Yaskawa INFORM job: X2_57-69(1)(90,0).JBI

/JOB
//NAME X2_57-69(1)(90,0)
//POS
///NPOS 359,359,359,20,0,0
///TOOL 0
///POSTYPE PULSE
///PULSE
C00000=1941,-102693,-129564,10,101994,-18
C00001=-114160,-110711,-132276,13468,99543,32658
C00002=-115352,64839,21503,33302,71092,28193
C00003=-108531,78392,43986,16123,55140,37786
C00004=-108866,85252,55178,17040,51979,37122
C00005=-108996,88365,60166,17472,50599,36819
C00006=-108995,88536,62039,17737,49581,36632
C00007=-109034,88718,61766,17697,49840,36662
C00008=-109565,92254,66229,18307,49070,36272
C00009=-109034,88718,61766,17697,49840,36662
C00010=-108904,85509,56654,17244,51243,36976
C00011=-108571,78466,45235,16289,54445,37659
C00012=-107997,64928,29160,15382,57165,38310
C00013=-122208,49017,56535,29995,44799,-20500
C00014=-121054,58896,69591,30976,41821,-21001
C00015=-120607,61403,73283,31313,40811,-21157
C00016=-120607,63170,76793,32085,39739,-21613
C00017=-120607,62274,75028,31694,40274,-21383
C00018=-120608,64965,78215,32056,39778,-21596
C00019=-120607,62274,75028,31694,40274,-21383
C00020=-121364,56707,67057,30894,42308,-20982
C00021=-122534,47142,54464,30007,45185,-20534
C00022=-121995,48000,54847,25969,42983,-17450
C00023=-121016,58047,68030,26856,40021,-17900
C00024=-120639,62684,74202,27406,38635,-18182
C00025=-120639,64991,78769,28376,37190,-18734
C00026=-120639,62684,74202,27406,38635,-18182
C00027=-120856,61874,74409,27857,38220,-18464
C00028=-120445,66454,79858,28202,37199,-18614
C00029=-120856,61874,74409,27857,38220,-18464
C00030=-121238,57224,68232,27288,39602,-18174
C00031=-122229,47153,55046,26369,42553,-17714
C00032=-125892,1211,1187,22441,56600,-15676
C00033=-137814,-110158,-69296,24031,60757,-19595
C00034=-137728,-112604,-73316,23755,61850,-19313
C00035=-105364,-57557,-72999,2137,103390,46474
C00036=-118914,16972,-18491,2200,108489,41969
C00037=-119887,15858,-15574,2165,106148,41596
C00038=-121510,15333,-13660,2144,104740,41021
C00039=-121541,15180,-12957,2137,104232,41000
C00040=-120276,15500,-14332,2152,105210,41447
C00041=-120275,15157,-12943,2141,104179,41429
C00042=-120845,15149,-12950,2139,104194,41236
C00043=-120275,15157,-12943,2141,104179,41429
C00044=-120276,15500,-14332,2152,105210,41447
C00045=-118914,16972,-18491,2200,108489,41969
C00046=-118859,16942,-18519,2200,108489,41988
C00047=-119832,15826,-15604,2165,106148,41615
C00048=-121413,15318,-13781,2144,104807,41053
C00049=-121413,15142,-12992,2137,104231,41043
C00050=-120221,15467,-14363,2153,105210,41465
C00051=-120221,15224,-12881,2141,104174,41447
C00052=-120790,15216,-12889,2139,104189,41254
C00053=-120221,15224,-12881,2141,104174,41447
C00054=-120221,15467,-14363,2153,105210,41465
C00055=-118859,16942,-18519,2200,108489,41988
C00056=-102402,-48698,-67991,2144,104784,47502
C00057=-177118,-86899,-49314,70294,69346,55717
C00058=-162665,-62437,-38431,68363,61957,60420
C00059=-158949,-60049,-34374,68890,58994,60353
C00060=-157479,-59004,-32692,69121,57826,60324
C00061=-157483,-57954,-30366,69642,57492,59876
C00062=-157504,-58291,-30998,69516,57587,59981
C00063=-155795,-59629,-31689,69630,56353,60099
C00064=-157504,-58291,-30998,69516,57587,59981
C00065=-157484,-58197,-30924,69514,57575,59985
C00066=-156523,-55844,-29677,69224,57103,60350
C00067=-157484,-58197,-30924,69514,57575,59985
C00068=-162670,-61686,-36716,68690,61698,60098
C00069=-161856,-67053,-41033,60813,38521,63477
C00070=-158996,-62210,-35558,60803,36300,63693
C00071=-157898,-60236,-33315,60834,35435,63760
C00072=-157901,-59173,-30986,61942,34994,63152
C00073=-156769,-58533,-30874,61190,34419,63655
C00074=-156166,-58108,-30651,60848,34087,63889
C00075=-156769,-58791,-31436,60917,34526,63803
C00076=-161883,-66170,-39058,61667,38156,62985
C00077=-175307,-91794,-54277,68294,45083,57713
C00078=-192656,-55134,-37587,64210,60039,59083
C00079=-162159,-23717,-10104,69718,77823,43469
C00080=-159534,-21701,-5637,70155,75421,43047
C00081=-158490,-20805,-3772,70360,74468,42873
C00082=-158493,-19842,-1317,70611,74104,42419
C00083=-158430,-19960,-1760,70561,74138,42521
C00084=-157077,-18912,-994,70615,73251,42719
C00085=-158430,-19960,-1760,70561,74138,42521
C00086=-162097,-22978,-8198,69866,77487,43129
C00087=-164656,-6441,2331,68796,80646,40119
C00088=-162354,-4355,7073,69146,78392,39620
C00089=-161441,-2725,10948,69469,77194,39063
C00090=-161443,-1987,12871,69626,76894,38710
C00091=-161439,-2551,11387,69503,77124,38984
C00092=-160415,-1923,12464,69637,76311,38965
C00093=-159548,-1589,12743,69678,75730,39076
C00094=-160719,-2768,10769,69490,76742,39193
C00095=-164702,-5497,5223,68969,80178,39553
C00096=-192656,-55134,-37587,64210,60039,59083
C00097=-125486,-104854,-75041,22917,86800,-65584
C00098=-126033,-92220,-87194,23391,99857,-63257
C00099=-126008,-87407,-69757,22927,92227,-64737
C00100=-122771,-89042,-67284,23124,89141,-64144
C00101=-121425,-89554,-66224,23215,87919,-63888
C00102=-121418,-87602,-63818,23218,87477,-63971
C00103=-121371,-87768,-64101,23220,87545,-63941
C00104=-119041,-87737,-64090,23370,86898,-63214
C00105=-121371,-87768,-64101,23220,87545,-63941
C00106=-119842,-88584,-64995,23320,87236,-63441
C00107=-119807,-91269,-65466,23334,86221,-63626
C00108=-119842,-88584,-64995,23320,87236,-63441
C00109=-121199,-88128,-66077,23230,88448,-63702
C00110=-124465,-86636,-68609,23034,91510,-64308
C00111=-142854,-85767,-72329,35934,81198,-48667
C00112=-140267,-86079,-63689,45810,58760,-32657
C00113=-135996,-80956,-60126,44498,56909,-31284
C00114=-134384,-78850,-58646,43955,56229,-30750
C00115=-134256,-77036,-56222,44175,55757,-30924
C00116=-134288,-77408,-56713,44133,55854,-30891
C00117=-132164,-77894,-56932,43544,54718,-30303
C00118=-134288,-77408,-56713,44133,55854,-30891
C00119=-88320,-91033,-56979,-46001,31828,15275
C00120=-89280,-88900,-56774,-44237,32046,14267
C00121=-88320,-91033,-56979,-46001,31828,15275
C00122=-85210,-101515,-62011,-50678,31900,18023
C00123=-89666,-105996,-71374,-46997,57370,39665
C00124=-112926,-92756,-65130,-39557,61499,44934
C00125=-117841,-88867,-61535,-38560,59130,43528
C00126=-119732,-87223,-60045,-38129,58240,42969
C00127=-119742,-85223,-57591,-38309,57852,43124
C00128=-119765,-85676,-58172,-38256,57941,43076
C00129=-121812,-86923,-58375,-37936,56635,42605
C00130=-119765,-85676,-58172,-38256,57941,43076
C00131=-121275,-85554,-58782,-37706,57631,42461
C00132=-122404,-83336,-58379,-37071,57860,41818
C00133=-121275,-85554,-58782,-37706,57631,42461
C00134=-114616,-91226,-63955,-39185,60786,44412
C00135=-114645,-97965,-79407,-37345,65578,42515
C00136=-116729,-83918,-76551,-18553,86191,61698
C00137=-117159,-89242,-76095,-11181,89587,70256
C00138=-119083,-90759,-73003,-11190,86687,69852
C00139=-119889,-89726,-70248,-11201,85432,69686
C00140=-119897,-88175,-68603,-11203,85218,69702
C00141=-119889,-89726,-70248,-11201,85432,69686
C00142=-119873,-91603,-70614,-11208,84708,69757
C00143=-119889,-89726,-70248,-11201,85432,69686
C00144=-107060,-93796,-69139,-19617,83326,67746
C00145=-109561,-94345,-69347,-19648,82582,66969
C00146=-107060,-93796,-69139,-19617,83326,67746
C00147=-120981,-91693,-72872,-11196,85873,69270
C00148=-118990,-90334,-76042,-11186,88750,69699
C00149=-119015,-93571,-89875,-11280,95471,69085
C00150=-121827,-98987,-110994,4235,90756,33976
C00151=-126467,-111869,-98615,30475,51467,-26148
C00152=-122938,-103029,-94111,27808,51796,-24337
C00153=-121643,-99583,-92275,26825,51945,-23680
C00154=-121634,-97826,-90039,26985,51518,-23798
C00155=-121643,-99583,-92275,26825,51945,-23680
C00156=-130783,-80407,-84869,35916,67887,-27578
C00157=-128717,-80853,-85070,35145,66956,-27002
C00158=-130783,-80407,-84869,35916,67887,-27578
C00159=-107674,-109601,-92730,7088,37825,-14001
C00160=-108083,-105924,-92018,7248,39302,-14088
C00161=-107674,-109601,-92730,7088,37825,-14001
C00162=-110011,-124661,-99237,10171,34381,-15732
C00163=-126906,-107253,-113226,22382,79753,-37979
C00164=-126893,-93432,-102362,29867,101882,-55415
C00165=-122864,-96655,-100816,29402,98217,-54829
C00166=-121215,-97700,-100096,29236,96792,-54563
C00167=-121210,-96197,-97952,29195,96310,-54685
C00168=-121215,-97700,-100096,29236,96792,-54563
C00169=-121163,-96448,-98340,29200,96390,-54646
C00170=-118846,-96389,-98319,29071,95614,-53959
C00171=-121163,-96448,-98340,29200,96390,-54646
C00172=-120263,-97948,-99498,29148,96030,-54394
C00173=-120240,-102374,-100607,29046,94623,-54741
C00174=-120263,-97948,-99498,29148,96030,-54394
C00175=-125973,-93962,-101877,29758,101067,-55277
C00176=-118596,-129181,-126473,-9366,77401,-2206
C00177=-114435,-108672,-97735,-33612,57488,30842
C00178=-118529,-101099,-93472,-31282,56999,29098
C00179=-120051,-98101,-91728,-30387,56847,28447
C00180=-120058,-96382,-89499,-30544,56421,28577
C00181=-120051,-98101,-91728,-30387,56847,28447
C00182=-120087,-96650,-89858,-30501,56482,28544
C00183=-122421,-96636,-89851,-29327,55655,27727
C00184=-120087,-96650,-89858,-30501,56482,28544
C00185=-120936,-97217,-90733,-29999,56393,28182
C00186=-120939,-93406,-89800,-29561,57600,27814
C00187=-120936,-97217,-90733,-29999,56393,28182
C00188=-115418,-107792,-96770,-33217,56982,30555
C00189=-105146,-130010,-122753,-24377,88875,54529
C00190=-114428,-145611,-119705,-15408,97435,71230
C00191=-117464,-150573,-117642,-15685,93169,70698
C00192=-118771,-152166,-116683,-15828,91559,70446
C00193=-118800,-148516,-114162,-15837,91865,70397
C00194=-118771,-152166,-116683,-15828,91559,70446
C00195=-89023,-160145,-112498,-25773,88935,79257
C00196=-92598,-162169,-112911,-26414,87133,78351
C00197=-89023,-160145,-112498,-25773,88935,79257
C00198=-143634,-123316,-108912,-7172,105756,63537
C00199=-144414,-127929,-109749,-7250,103844,63374
C00200=-143634,-123316,-108912,-7172,105756,63537
C00201=-142718,-121013,-109514,-7059,107379,63770
C00202=-140567,-114497,-110685,-6827,111603,64303
C00203=-106156,-132360,-130153,-17350,90664,54849
C00204=-113451,-107662,-104229,-36971,70393,33800
C00205=-118206,-101735,-100389,-35240,68968,32234
C00206=-120007,-99320,-98805,-34543,68461,31631
C00207=-120014,-97721,-96632,-34652,68030,31771
C00208=-120007,-99320,-98805,-34543,68461,31631
C00209=-120011,-97828,-96896,-34630,68120,31742
C00210=-122349,-97818,-96890,-33771,67193,31043
C00211=-120011,-97828,-96896,-34630,68120,31742
C00212=-121054,-97492,-97790,-34094,68307,31234
C00213=-121054,-93214,-96669,-33787,69569,30828
C00214=-121054,-97492,-97790,-34094,68307,31234
C00215=-114636,-105862,-103272,-36519,70163,33365
C00216=-114279,-101889,-100082,-25331,80876,44864
C00217=-118566,-99424,-96391,-24445,78685,43735
C00218=-120245,-97521,-93811,-24102,77637,43327
C00219=-120247,-96657,-92660,-24122,77395,43376
C00220=-120219,-96976,-93108,-24119,77505,43364
C00221=-122549,-96954,-93097,-23561,76842,42630
C00222=-120219,-96976,-93108,-24119,77505,43364
C00223=-114306,-100541,-98340,-25348,80523,44930
C00224=-120621,-97394,-101621,-24202,63073,45941
C00225=-120621,-97613,-99404,-24510,61722,46250
C00226=-126885,-95808,-100508,-15136,62705,44325
C00227=-124891,-100138,-106487,-19050,76932,40471
C00228=-124330,-97085,-92322,-20020,71587,41486
C00229=-120096,-97587,-96517,-20033,105608,38386
C00230=-120621,-97666,-97219,-19653,110159,37614
C00231=-120621,-97564,-100279,-19942,111985,37290
C00232=-114267,-119022,-117316,-18586,97333,41934
C00233=-120586,-140068,-100376,-59799,22791,77658
C00234=-120585,-131836,-89399,-65340,21573,80326
C00235=-120301,-131910,-88922,-66286,21610,80804
C00236=-120198,-131934,-88749,-66625,21626,80975
C00237=-119916,-129593,-85873,-68118,21579,81715
C00238=-118482,-138777,-95380,-52510,29730,72880
C00239=-120255,-147562,-109916,-33672,49046,60189
C00240=-120254,-140089,-100414,-34669,47370,60868
C00241=-115468,-148569,-111904,-12737,99323,53877
C00242=-120588,-148294,-110670,-9262,106248,51768
C00243=-120588,-160541,-124626,-9395,108516,51590
C00244=-136842,-121669,-124376,16041,91150,-8624
C00245=-120606,-113410,-86554,36159,18075,-56282
C00246=-120605,-110678,-81352,39700,16640,-57934
C00247=-120584,-111701,-82271,39578,16661,-57878
C00248=-120580,-111920,-82466,39553,16665,-57867
C00249=-120605,-109556,-79302,41216,16112,-58638
C00250=-124077,-125780,-98632,32708,39047,-51685
C00251=-120496,-124050,-111043,24637,69959,-42697
C00252=-120664,-121871,-104765,25113,67511,-43309
C00253=-121671,-124094,-110510,20986,97112,-39569
C00254=-120608,-124256,-111795,20648,99670,-38855
C00255=-120609,-125131,-115147,20777,101183,-38590
C00256=-120610,-125783,-123647,21277,105768,-37763
C00257=-120668,-128769,-125921,-5871,89606,-827
C00258=-107053,-95803,-77707,-38578,68772,44507
C00259=-120618,-86239,-59568,-37363,57829,42393
C00260=-120528,-85716,-59123,-36997,58097,42691
C00261=-120619,-91352,-71155,-22510,73817,56639
C00262=-119738,-88100,-63683,-22964,71349,57460
C00263=-119548,-88867,-66660,-18371,78749,62657
C00264=-120622,-86591,-69531,-13569,88626,68335
C00265=-120425,-89920,-79314,-13611,92853,67941
C00266=-120620,-95688,-83779,-13612,92610,67900
C00267=-120653,-118153,-99445,8937,69074,27704
C00268=-120618,-86290,-59555,39610,31833,-26802
C00269=-120617,-83679,-54099,41791,30283,-27941
C00270=-120617,-83181,-53105,42201,30015,-28153
C00271=-120617,-83020,-52785,42335,29929,-28222
C00272=-120619,-93115,-75724,25664,64689,-43944
C00273=-120826,-86244,-59129,27057,59793,-46292
C00274=-121400,-88637,-64040,23275,84750,-62478
C00275=-120618,-88758,-64988,22876,88456,-64391
C00276=-120618,-90407,-68808,22886,89847,-64125
C00277=-120645,-96149,-85177,23134,96436,-62865
C00278=-120704,-139648,-98792,22953,83536,-65363
C00279=-201677,-83839,-16745,82551,61455,23328
C00280=-193287,-71994,-23753,71338,80116,26125
C00281=-188716,-68676,-18939,72756,76807,26050
C00282=-186807,-37234,2063,68557,93943,25131
C00283=-186791,-37375,1977,68560,93924,25125
C00284=-188875,-55332,-8770,71294,85660,29887
C00285=-186990,-46090,-3659,67979,93495,33535
C00286=-187169,-52287,-8326,67185,92343,33510
C00287=-188906,-62105,-11935,69333,88967,33384
C00288=-188683,-64142,-13243,69128,88603,33879
C00289=-187867,-62779,-12578,68415,90081,34352
C00290=-188794,-66315,-17993,66765,90030,34259
C00291=-197371,-61565,-20436,64467,96999,34726
C00292=-180892,-45026,-152,77390,64230,28169
C00293=-201677,-83839,-16745,82551,61455,23328
C00294=-102465,-98091,-57376,11154,53691,1192
C00295=-117523,-2788,-9530,25488,75365,-1139
C00296=-125139,57134,55592,35785,69072,-6421
C00297=-125133,64451,72830,37508,63513,-8429
C00298=-123932,76756,90632,38887,59314,-9544
C00299=-123464,84249,101464,39928,56909,-10353
C00300=-122296,71715,85090,35181,54513,-6915
C00301=-122189,68599,81314,33173,52324,-4280
C00302=-122589,68250,80867,31901,50792,-2732
C00303=-122908,67120,79438,30365,49475,-1044
C00304=-123218,66439,78655,28729,48083,651
C00305=-123718,66653,78885,28024,47440,1365
C00306=-121882,59213,71115,24134,43656,7775
C00307=-110842,52453,67135,-14467,33841,33723
C00308=-111073,52381,67059,-14368,33810,33647
C00309=-110346,48653,61790,-14496,35224,33792
C00310=-108666,36587,42456,-14007,41045,33643
C00311=-114621,109196,43725,31616,85766,30078
C00312=-108492,104701,44017,11484,73458,41705
C00313=-108890,108743,52585,11893,70378,41274
C00314=-108566,112524,59213,11878,68242,41168
C00315=-105655,126679,78153,10634,63557,41739
C00316=-105456,124563,73948,10396,65010,41943
C00317=-114621,109196,43725,31616,85766,30078
C00318=-117523,-2788,-9530,25488,75365,-1139
C00319=-102465,-98091,-57376,11154,53691,1192
C00320=-194924,-89332,-18186,86283,57168,22588
C00321=-189291,-99620,-43569,70052,49879,58298
C00322=-183385,-95654,-38841,71457,45923,58650
C00323=-179289,-94967,-37057,72626,43143,58783
C00324=-180541,-94166,-36956,72139,44032,58817
C00325=-181760,-88303,-31492,78702,40431,52425
C00326=-191947,-67176,-20621,75434,55592,47212
C00327=-188895,-71260,-14971,91913,47690,32624
C00328=-190378,-73018,-17241,90953,48654,32921
C00329=-194954,-78245,-22550,88961,51649,33203
C00330=-209629,-115340,-51402,66324,56026,36469
C00331=-117179,-93991,-70029,-10923,64438,-31948
C00332=-91116,-86743,-69135,-16598,71993,-23160
C00333=-103770,-45855,-47036,-2494,89723,45807
C00334=-105440,-45139,-42797,-2405,87433,45286
C00335=-105872,-44623,-40732,-2383,86415,45158
C00336=-107998,-22692,-26100,-2267,88615,44398
C00337=-107613,-23106,-28265,-2289,89747,44508
C00338=-106174,-23599,-32412,-2371,92085,44950
C00339=-103769,-45855,-47037,-2494,89723,45807
C00340=-105440,-45140,-42797,-2405,87433,45286
C00341=-105983,-45111,-40907,-2377,86269,45123
C00342=-108050,-23400,-26513,-2264,88505,44381
C00343=-107613,-23106,-28265,-2289,89747,44508
C00344=-106174,-23599,-32412,-2371,92085,44950
C00345=-106187,-23536,-40664,-2395,97191,44849
C00346=-112777,14050,-22213,-10109,94464,-2996
C00347=-124710,91382,43994,-20502,78853,-68751
C00348=-124710,90699,45107,-20567,77880,-68584
C00349=-124711,89465,47608,-20728,75840,-68228
C00350=-124762,93463,53735,-20858,74219,-67960
C00351=-124700,97572,58988,-20989,73184,-67752
C00352=-127201,90948,48694,-14686,76522,-68030
C00353=-125335,102453,72014,-19381,53758,-65341
C00354=-124858,91287,58679,-21278,49111,-64908
C00355=-124711,88619,50210,-21147,50008,-65361
C00356=-120351,15313,-32439,-6340,69848,-64116
C00357=-119749,-104989,-49747,-18878,19546,-56964
C00358=1074,-84890,-111921,820,92639,-133
BC00000=210618,668760,578653
BC00001=307087,668760,191900
BC00002=307087,789553,191900
BC00003=307087,789553,191900
BC00004=307087,789553,191900
BC00005=307087,789553,191900
BC00006=307087,789553,191900
BC00007=307087,789553,191900
BC00008=307087,789553,191900
BC00009=307087,789553,191900
BC00010=307087,789553,191900
BC00011=307087,789553,191900
BC00012=307087,789553,191900
BC00013=319173,776954,280603
BC00014=319173,776954,280603
BC00015=319173,776954,280603
BC00016=319173,776954,280603
BC00017=319173,776954,280603
BC00018=319173,776954,280603
BC00019=319173,776954,280603
BC00020=319173,776954,280603
BC00021=319173,776954,280603
BC00022=324465,771616,271785
BC00023=324465,771616,271785
BC00024=324465,771616,271785
BC00025=324465,771616,271785
BC00026=324465,771616,271785
BC00027=324465,771616,271785
BC00028=324465,771616,271785
BC00029=324465,771616,271785
BC00030=324465,771616,271785
BC00031=324465,771616,271785
BC00032=324465,747237,368530
BC00033=324465,670069,674761
BC00034=169071,670069,459913
BC00035=137209,684775,182974
BC00036=137209,684775,182974
BC00037=137209,684775,182974
BC00038=137209,684775,182974
BC00039=137209,684775,182974
BC00040=137209,684775,182974
BC00041=137209,684775,182974
BC00042=137209,684775,182974
BC00043=137209,684775,182974
BC00044=137209,684775,182974
BC00045=137209,684775,182974
BC00046=136881,731969,182759
BC00047=136881,731969,182759
BC00048=136881,731969,182759
BC00049=136881,731969,182759
BC00050=136881,731969,182759
BC00051=136881,731969,182759
BC00052=136881,731969,182759
BC00053=136881,731969,182759
BC00054=136881,731969,182759
BC00055=136881,731969,182759
BC00056=136881,673536,182759
BC00057=33003,666220,204314
BC00058=33003,666220,204314
BC00059=33003,666220,204314
BC00060=33003,666220,204314
BC00061=33003,666220,204314
BC00062=33003,666220,204314
BC00063=33003,666220,204314
BC00064=33003,666220,204314
BC00065=33003,666220,204314
BC00066=33003,666220,204314
BC00067=33003,666220,204314
BC00068=33003,666220,204314
BC00069=48470,666220,217137
BC00070=48470,666220,217137
BC00071=48470,666220,217137
BC00072=48470,666220,217137
BC00073=48470,666220,217137
BC00074=48470,666220,217137
BC00075=48470,666220,217137
BC00076=48470,666220,217137
BC00077=48470,666220,217137
BC00078=48470,666220,217137
BC00079=15,666220,230034
BC00080=15,666220,230034
BC00081=15,666220,230034
BC00082=15,666220,230034
BC00083=15,666220,230034
BC00084=15,666220,230034
BC00085=15,666220,230034
BC00086=15,666220,230034
BC00087=15,666220,235835
BC00088=15,666220,235835
BC00089=15,666220,235835
BC00090=15,666220,235835
BC00091=15,666220,235835
BC00092=15,666221,235834
BC00093=15,666220,235835
BC00094=15,666220,235835
BC00095=15,666220,235835
BC00096=48470,666220,217137
BC00097=32831,670161,1075175
BC00098=32831,729596,1075175
BC00099=32831,729596,1075175
BC00100=32831,729596,1075175
BC00101=32831,729596,1075175
BC00102=32831,729596,1075175
BC00103=32831,729596,1075175
BC00104=32831,729596,1075175
BC00105=32831,729596,1075175
BC00106=32831,729596,1075175
BC00107=32831,729596,1075175
BC00108=32831,729596,1075175
BC00109=32831,729596,1075175
BC00110=32831,729596,1075175
BC00111=37728,721693,1075175
BC00112=41810,715107,1075175
BC00113=41810,715107,1075175
BC00114=41810,715107,1075175
BC00115=41810,715107,1075175
BC00116=41810,715107,1075175
BC00117=41810,715107,1075175
BC00118=41810,715107,1075175
BC00119=41810,715107,1075175
BC00120=41810,715107,1075175
BC00121=41810,715107,1075175
BC00122=41810,715107,1075175
BC00123=53876,706752,1075175
BC00124=60427,702216,1075175
BC00125=60427,702216,1075175
BC00126=60427,702216,1075175
BC00127=60427,702216,1075175
BC00128=60427,702216,1075175
BC00129=60427,702216,1075175
BC00130=60427,702216,1075175
BC00131=60427,702216,1075175
BC00132=60427,702216,1075175
BC00133=60427,702216,1075175
BC00134=60427,702216,1075175
BC00135=60427,702216,1075175
BC00136=46834,716034,1075175
BC00137=41397,721561,1075175
BC00138=41397,721561,1075175
BC00139=41397,721561,1075175
BC00140=41397,721561,1075175
BC00141=41397,721561,1075175
BC00142=41397,721561,1075175
BC00143=41397,721561,1075175
BC00144=41397,721561,1075175
BC00145=41397,721561,1075175
BC00146=41397,721561,1075175
BC00147=41397,721561,1075175
BC00148=41397,721561,1075175
BC00149=41397,721561,1075175
BC00150=77086,766277,1075175
BC00151=137161,841550,1075175
BC00152=137161,841550,1075175
BC00153=137161,841550,1075175
BC00154=137161,841550,1075175
BC00155=137161,841550,1075175
BC00156=137161,841550,1075175
BC00157=137161,841550,1075175
BC00158=137161,841550,1075175
BC00159=137161,841550,1075175
BC00160=137161,841550,1075175
BC00161=137161,841550,1075175
BC00162=137161,841550,1075175
BC00163=128673,864447,1075175
BC00164=121183,884651,1075175
BC00165=121183,884651,1075175
BC00166=121183,884651,1075175
BC00167=121183,884651,1075175
BC00168=121183,884651,1075175
BC00169=121183,884651,1075175
BC00170=121183,884651,1075175
BC00171=121183,884651,1075175
BC00172=121183,884651,1075175
BC00173=121183,884651,1075175
BC00174=121183,884651,1075175
BC00175=121183,884651,1075175
BC00176=162519,857645,1075175
BC00177=188050,840965,1075175
BC00178=188050,840965,1075175
BC00179=188050,840965,1075175
BC00180=188050,840965,1075175
BC00181=188050,840965,1075175
BC00182=188050,840965,1075175
BC00183=188050,840965,1075175
BC00184=188050,840965,1075175
BC00185=188050,840965,1075175
BC00186=188050,840965,1075175
BC00187=188050,840965,1075175
BC00188=188050,840965,1075175
BC00189=177981,881480,1075175
BC00190=169709,914761,1075175
BC00191=169709,914761,1075175
BC00192=169709,914761,1075175
BC00193=169709,914761,1075175
BC00194=169709,914761,1075175
BC00195=169709,914761,1075175
BC00196=169709,914761,1075175
BC00197=169709,914761,1075175
BC00198=169709,914761,1075175
BC00199=169709,914761,1075175
BC00200=169709,914761,1075175
BC00201=169709,914761,1075175
BC00202=169709,914761,1075175
BC00203=159152,880596,1075175
BC00204=150354,852125,1075175
BC00205=150354,852125,1075175
BC00206=150354,852125,1075175
BC00207=150354,852125,1075175
BC00208=150354,852125,1075175
BC00209=150354,852125,1075175
BC00210=150354,852125,1075175
BC00211=150354,852125,1075175
BC00212=150354,852125,1075175
BC00213=150354,852125,1075175
BC00214=150354,852125,1075175
BC00215=150354,852125,1075175
BC00216=138535,800539,1075175
BC00217=138535,800539,1075175
BC00218=138535,800539,1075175
BC00219=138535,800539,1075175
BC00220=138535,800539,1075175
BC00221=138535,800539,1075175
BC00222=138535,800539,1075175
BC00223=138535,800539,1075175
BC00224=139926,838224,1075175
BC00225=134477,841860,1075175
BC00226=132297,843314,1075175
BC00227=135301,861824,1075175
BC00228=135628,791701,1075175
BC00229=127557,845014,1075175
BC00230=128457,853081,1075175
BC00231=133547,854476,1075175
BC00232=133547,854476,1075175
BC00233=185526,847143,1075175
BC00234=185547,847145,1075175
BC00235=180367,852195,1075175
BC00236=178499,854016,1075175
BC00237=178499,854016,1075175
BC00238=181436,863252,1075175
BC00239=187425,882089,1075175
BC00240=187544,843803,1075173
BC00241=163075,924936,1075175
BC00242=160150,941259,1075175
BC00243=163894,945401,1075175
BC00244=155016,866117,1075175
BC00245=147551,828920,1075175
BC00246=147562,828921,1075175
BC00247=152516,835936,1075175
BC00248=153570,837428,1075175
BC00249=153570,837428,1075175
BC00250=143866,860842,1075175
BC00251=131316,891124,1075175
BC00252=131456,861099,1075175
BC00253=136555,907393,1075175
BC00254=134846,911418,1075175
BC00255=129544,912127,1075175
BC00256=129523,912125,1075175
BC00257=99118,813312,1075175
BC00258=64307,700180,1075175
BC00259=58098,703250,1075175
BC00260=55325,704971,1075175
BC00261=41598,728447,1075175
BC00262=60495,698876,1075175
BC00263=53827,709917,1075175
BC00264=47010,724325,1075175
BC00265=50143,727052,1075175
BC00266=50122,727050,1075175
BC00267=43900,716168,1075175
BC00268=35524,701519,1075175
BC00269=35534,701520,1075175
BC00270=39202,708199,1075175
BC00271=40669,710870,1075175
BC00272=31604,749687,1075172
BC00273=32090,681060,1075175
BC00274=35435,723771,1075175
BC00275=34090,730815,1075175
BC00276=29574,733664,1075175
BC00277=29574,733664,1075175
BC00278=29574,668853,1075175
BC00279=15,675786,401985
BC00280=15,747285,294679
BC00281=15,747285,294679
BC00282=15,747285,294679
BC00283=15,747285,294679
BC00284=15,747285,294679
BC00285=15,747285,294679
BC00286=15,747285,294679
BC00287=15,747285,294679
BC00288=15,747285,294679
BC00289=15,747285,294679
BC00290=15,747285,294679
BC00291=15,747285,294679
BC00292=15,675786,401985
BC00293=15,675786,401985
BC00294=281438,669247,530529
BC00295=311998,746592,376004
BC00296=327524,785889,297495
BC00297=327524,785889,297495
BC00298=327524,785889,297495
BC00299=327524,785889,297495
BC00300=327524,785889,297495
BC00301=327524,785889,297495
BC00302=327524,785889,297495
BC00303=327524,785889,297495
BC00304=327524,785889,297495
BC00305=327524,785889,297495
BC00306=327524,785889,297495
BC00307=327524,785889,297495
BC00308=327524,785889,297495
BC00309=327524,785889,297495
BC00310=327524,785889,297495
BC00311=301537,784116,209
BC00312=301537,784116,209
BC00313=301537,784116,209
BC00314=301537,784116,209
BC00315=301537,784116,209
BC00316=301537,784116,209
BC00317=301537,784116,209
BC00318=311998,746592,376004
BC00319=281438,669247,530529
BC00320=28742,675786,401985
BC00321=69504,715923,290542
BC00322=69504,715923,290542
BC00323=69504,715923,290542
BC00324=69504,715923,290542
BC00325=69504,715923,290542
BC00326=69504,715923,290542
BC00327=69504,715923,290542
BC00328=69504,715923,290542
BC00329=69504,715923,290542
BC00330=69504,715923,290542
BC00331=108267,707570,269586
BC00332=108267,707570,269586
BC00333=115634,729988,290459
BC00334=115634,729988,290459
BC00335=115634,729988,290459
BC00336=115634,729988,290459
BC00337=115634,729988,290459
BC00338=115634,729988,290459
BC00339=115460,777038,290246
BC00340=115460,777038,290246
BC00341=115460,777038,290246
BC00342=115460,777038,290246
BC00343=115460,777038,290246
BC00344=115460,777038,290246
BC00345=115460,777038,290246
BC00346=136842,705148,185844
BC00347=166172,670726,41167
BC00348=166193,670728,53
BC00349=164826,672048,53
BC00350=164280,672575,53
BC00351=164280,672575,53
BC00352=163972,755654,53
BC00353=160957,747196,53
BC00354=159846,741879,53
BC00355=160544,735428,53
BC00356=166172,670726,41167
BC00357=166172,670726,387185
BC00358=166172,670726,387185
EC00000=798156,0
EC00001=798156,0
EC00002=798156,0
EC00003=798156,0
EC00004=798156,0
EC00005=798156,0
EC00006=798156,0
EC00007=798156,0
EC00008=798156,0
EC00009=798156,0
EC00010=798156,0
EC00011=798156,0
EC00012=798156,0
EC00013=798156,0
EC00014=798156,0
EC00015=798156,0
EC00016=798156,0
EC00017=798156,0
EC00018=798156,0
EC00019=798156,0
EC00020=798156,0
EC00021=798156,0
EC00022=798156,0
EC00023=798156,0
EC00024=798156,0
EC00025=798156,0
EC00026=798156,0
EC00027=798156,0
EC00028=798156,0
EC00029=798156,0
EC00030=798156,0
EC00031=798156,0
EC00032=798156,0
EC00033=798156,0
EC00034=798156,0
EC00035=798156,0
EC00036=798156,0
EC00037=798156,0
EC00038=798156,0
EC00039=798156,0
EC00040=798156,0
EC00041=798156,0
EC00042=798156,0
EC00043=798156,0
EC00044=798156,0
EC00045=798156,0
EC00046=798156,0
EC00047=798156,0
EC00048=798156,0
EC00049=798156,0
EC00050=798156,0
EC00051=798156,0
EC00052=798156,0
EC00053=798156,0
EC00054=798156,0
EC00055=798156,0
EC00056=798156,0
EC00057=798156,0
EC00058=798156,0
EC00059=798156,0
EC00060=798156,0
EC00061=798156,0
EC00062=798156,0
EC00063=798156,0
EC00064=798156,0
EC00065=798156,0
EC00066=798156,0
EC00067=798156,0
EC00068=798156,0
EC00069=798156,0
EC00070=798156,0
EC00071=798156,0
EC00072=798156,0
EC00073=798156,0
EC00074=798156,0
EC00075=798156,0
EC00076=798156,0
EC00077=798156,0
EC00078=798156,0
EC00079=798156,0
EC00080=798156,0
EC00081=798156,0
EC00082=798156,0
EC00083=798156,0
EC00084=798156,0
EC00085=798156,0
EC00086=798156,0
EC00087=798156,0
EC00088=798156,0
EC00089=798156,0
EC00090=798156,0
EC00091=798156,0
EC00092=798155,0
EC00093=798156,0
EC00094=798156,0
EC00095=798156,0
EC00096=798156,0
EC00097=975524,0
EC00098=975524,0
EC00099=975524,0
EC00100=975524,0
EC00101=975524,0
EC00102=975524,0
EC00103=975524,0
EC00104=975524,0
EC00105=975524,0
EC00106=975524,0
EC00107=975524,0
EC00108=975524,0
EC00109=975524,0
EC00110=975524,0
EC00111=975524,0
EC00112=975524,0
EC00113=975524,0
EC00114=975524,0
EC00115=975524,0
EC00116=975524,0
EC00117=975524,0
EC00118=975524,0
EC00119=975524,0
EC00120=975524,0
EC00121=975524,0
EC00122=975524,0
EC00123=975524,0
EC00124=975524,0
EC00125=975524,0
EC00126=975524,0
EC00127=975524,0
EC00128=975524,0
EC00129=975524,0
EC00130=975524,0
EC00131=975524,0
EC00132=975524,0
EC00133=975524,0
EC00134=975524,0
EC00135=975524,0
EC00136=975524,0
EC00137=975524,0
EC00138=975524,0
EC00139=975524,0
EC00140=975524,0
EC00141=975524,0
EC00142=975524,0
EC00143=975524,0
EC00144=975524,0
EC00145=975524,0
EC00146=975524,0
EC00147=975524,0
EC00148=975524,0
EC00149=975524,0
EC00150=975524,0
EC00151=975524,0
EC00152=975524,0
EC00153=975524,0
EC00154=975524,0
EC00155=975524,0
EC00156=975524,0
EC00157=975524,0
EC00158=975524,0
EC00159=975524,0
EC00160=975524,0
EC00161=975524,0
EC00162=975524,0
EC00163=975524,0
EC00164=975524,0
EC00165=975524,0
EC00166=975524,0
EC00167=975524,0
EC00168=975524,0
EC00169=975524,0
EC00170=975524,0
EC00171=975524,0
EC00172=975524,0
EC00173=975524,0
EC00174=975524,0
EC00175=975524,0
EC00176=975524,0
EC00177=975524,0
EC00178=975524,0
EC00179=975524,0
EC00180=975524,0
EC00181=975524,0
EC00182=975524,0
EC00183=975524,0
EC00184=975524,0
EC00185=975524,0
EC00186=975524,0
EC00187=975524,0
EC00188=975524,0
EC00189=975524,0
EC00190=975524,0
EC00191=975524,0
EC00192=975524,0
EC00193=975524,0
EC00194=975524,0
EC00195=975524,0
EC00196=975524,0
EC00197=975524,0
EC00198=975524,0
EC00199=975524,0
EC00200=975524,0
EC00201=975524,0
EC00202=975524,0
EC00203=975524,0
EC00204=975524,0
EC00205=975524,0
EC00206=975524,0
EC00207=975524,0
EC00208=975524,0
EC00209=975524,0
EC00210=975524,0
EC00211=975524,0
EC00212=975524,0
EC00213=975524,0
EC00214=975524,0
EC00215=975524,0
EC00216=975524,0
EC00217=975524,0
EC00218=975524,0
EC00219=975524,0
EC00220=975524,0
EC00221=975524,0
EC00222=975524,0
EC00223=975524,0
EC00224=975524,0
EC00225=975524,0
EC00226=975524,0
EC00227=975524,0
EC00228=975524,0
EC00229=975524,0
EC00230=975524,0
EC00231=975524,0
EC00232=975524,0
EC00233=975524,0
EC00234=975524,0
EC00235=975524,0
EC00236=975524,0
EC00237=975524,0
EC00238=975524,0
EC00239=975524,0
EC00240=975522,1
EC00241=975524,0
EC00242=975524,0
EC00243=975524,0
EC00244=975524,0
EC00245=975524,0
EC00246=975524,0
EC00247=975524,0
EC00248=975524,0
EC00249=975524,0
EC00250=975524,0
EC00251=975524,0
EC00252=975524,0
EC00253=975524,0
EC00254=975524,0
EC00255=975524,0
EC00256=975524,0
EC00257=975524,0
EC00258=975524,0
EC00259=975524,0
EC00260=975524,0
EC00261=975524,0
EC00262=975524,0
EC00263=975524,0
EC00264=975524,0
EC00265=975524,0
EC00266=975524,0
EC00267=975524,0
EC00268=975524,0
EC00269=975524,0
EC00270=975524,0
EC00271=975524,0
EC00272=975522,1
EC00273=975524,0
EC00274=975524,0
EC00275=975524,0
EC00276=975524,0
EC00277=975524,0
EC00278=975524,0
EC00279=798156,0
EC00280=798156,0
EC00281=798156,0
EC00282=798156,0
EC00283=798156,0
EC00284=798156,0
EC00285=798156,0
EC00286=798156,0
EC00287=798156,0
EC00288=798156,0
EC00289=798156,0
EC00290=798156,0
EC00291=798156,0
EC00292=798156,0
EC00293=798156,0
EC00294=798156,0
EC00295=798156,0
EC00296=798156,0
EC00297=798156,0
EC00298=798156,0
EC00299=798156,0
EC00300=798156,0
EC00301=798156,0
EC00302=798156,0
EC00303=798156,0
EC00304=798156,0
EC00305=798156,0
EC00306=798156,0
EC00307=798156,0
EC00308=798156,0
EC00309=798156,0
EC00310=798156,0
EC00311=798156,0
EC00312=798156,0
EC00313=798156,0
EC00314=798156,0
EC00315=798156,0
EC00316=798156,0
EC00317=798156,0
EC00318=798156,0
EC00319=798156,0
EC00320=798156,0
EC00321=798156,0
EC00322=798156,0
EC00323=798156,0
EC00324=798156,0
EC00325=798156,0
EC00326=798156,0
EC00327=798156,0
EC00328=798156,0
EC00329=798156,0
EC00330=798156,0
EC00331=798156,0
EC00332=798156,0
EC00333=798156,0
EC00334=798156,0
EC00335=798156,0
EC00336=798156,0
EC00337=798156,0
EC00338=798156,0
EC00339=798156,0
EC00340=798156,0
EC00341=798156,0
EC00342=798156,0
EC00343=798156,0
EC00344=798156,0
EC00345=798156,0
EC00346=798156,0
EC00347=798156,0
EC00348=798156,0
EC00349=798156,0
EC00350=798156,0
EC00351=798156,0
EC00352=798156,0
EC00353=798156,0
EC00354=798156,0
EC00355=798156,0
EC00356=798156,0
EC00357=798156,0
EC00358=798156,0
///POSTYPE BASE
///RECTAN
///RCONF 0,0,0,0,0,0,0,0,0,0,0,0,0,0,0,0,0,0,0,0,0,0,0,0
P00006=0.222,-3.123,-1.508,0.0000,0.0000,0.0000
P00020=2.715,4.999,8.452,0.0000,0.0000,0.0000
P00021=-0.225,-6.128,-0.405,0.0000,0.0000,0.0000
P00022=0.222,-3.123,-1.508,0.0000,0.0000,0.0000
P00023=0.143,-0.036,0.682,0.0000,0.0000,0.0000
P00024=0.145,-0.552,1.326,0.0000,0.0000,0.0000
P00025=-2.003,0.006,0.728,0.0000,0.0000,0.0000
P00026=0.562,-0.002,-0.337,0.0000,0.0000,0.0000
P00031=1.853,-0.001,-1.549,0.0000,0.0000,0.0000
P00032=1.957,0.503,-7.217,0.0000,0.0000,0.0000
///RCONF 0,0,0,0,1,0,0,0,0,0,0,0,0,0,0,0,0,0,0,0,0,0,0,0
P00033=-0.123,0.612,-5.012,0.0000,0.0000,0.0000
///RCONF 0,0,0,0,0,0,0,0,0,0,0,0,0,0,0,0,0,0,0,0,0,0,0,0
P00034=-0.304,0.773,-2.693,0.0000,0.0000,0.0000
P00035=2.817,0.591,-1.622,0.0000,0.0000,0.0000
P00036=-1.108,-0.829,1.850,0.0000,0.0000,0.0000
P00037=0.023,0.937,-2.677,0.0000,0.0000,0.0000
P00038=0.158,-1.133,-1.952,0.0000,0.0000,0.0000
P00039=0.012,-3.081,-0.106,0.0000,0.0000,0.0000
P00040=-0.030,9.648,2.467,0.0000,0.0000,0.0000
P00041=0.192,3.924,0.305,0.0000,0.0000,0.0000
P00042=-0.217,1.941,0.413,0.0000,0.0000,0.0000
//INST
///DATE 2024/11/05 12:47
///ATTR SC,RW
///GROUP1 RB1,BS1
///GROUP2 ST1
NOP
'X2_57-69(1)(90,0)
'Down
'Down
MOVJ C00000 BC00000 VJ=100.00  +MOVJ EC00000 VJ=100.00
MOVJ C00001 BC00001 VJ=100.00  +MOVJ EC00001 VJ=100.00
MOVJ C00002 BC00002 VJ=100.00  +MOVJ EC00002 VJ=100.00
'Path S4672
SFTOF3D
MOVJ C00003 BC00003 VJ=100.00  +MOVJ EC00003 VJ=100.00
MOVL C00004 BC00004 V=800.0  +MOVJ EC00004 VJ=100.00
SMOVL C00005 BC00005 V=166.7  +MOVJ EC00005
SREFP 3 C00006 BC00006  +REFP EC00006
CALL JOB:SEARCH-R1-S13D
SET P020 P006
SFTON3D P020
SMOVL C00007 BC00007 V=166.7  +MOVJ EC00007
SREFP 3 C00008 BC00008  +REFP EC00008
CALL JOB:SEARCH-R1-S13D
SET P020 P006
SFTON3D P020
SMOVL C00009 BC00009 V=166.7  +MOVJ EC00009
MOVL C00010 BC00010 V=800.0  +MOVJ EC00010 VJ=100.00
MOVL C00011 BC00011 V=1000.0  +MOVJ EC00011 VJ=100.00
'EndPath S4672
'Path S4673
SFTOF3D
MOVJ C00012 BC00012 VJ=100.00  +MOVJ EC00012 VJ=100.00
MOVJ C00013 BC00013 VJ=100.00  +MOVJ EC00013 VJ=100.00
MOVL C00014 BC00014 V=800.0  +MOVJ EC00014 VJ=100.00
SMOVL C00015 BC00015 V=166.7  +MOVJ EC00015
SREFP 3 C00016 BC00016  +REFP EC00016
CALL JOB:SEARCH-R1-S13D
SET P021 P006
SFTON3D P021
SMOVL C00017 BC00017 V=166.7  +MOVJ EC00017
SREFP 3 C00018 BC00018  +REFP EC00018
CALL JOB:SEARCH-R1-S13D
SET P021 P006
SFTON3D P021
SMOVL C00019 BC00019 V=166.7  +MOVJ EC00019
MOVL C00020 BC00020 V=800.0  +MOVJ EC00020 VJ=100.00
MOVL C00021 BC00021 V=1000.0  +MOVJ EC00021 VJ=100.00
'EndPath S4673
'Path S4674
SFTOF3D
MOVJ C00022 BC00022 VJ=100.00  +MOVJ EC00022 VJ=100.00
MOVL C00023 BC00023 V=800.0  +MOVJ EC00023 VJ=100.00
SMOVL C00024 BC00024 V=166.7  +MOVJ EC00024
SREFP 3 C00025 BC00025  +REFP EC00025
CALL JOB:SEARCH-R1-S13D
SET P022 P006
SFTON3D P022
SMOVL C00026 BC00026 V=166.7  +MOVJ EC00026
SMOVL C00027 BC00027 V=166.7  +MOVJ EC00027
SREFP 3 C00028 BC00028  +REFP EC00028
CALL JOB:SEARCH-R1-S13D
SET P022 P006
SFTON3D P022
SMOVL C00029 BC00029 V=166.7  +MOVJ EC00029
MOVL C00030 BC00030 V=800.0  +MOVJ EC00030 VJ=100.00
MOVL C00031 BC00031 V=1000.0  +MOVJ EC00031 VJ=100.00
'EndPath S4674
MOVJ C00032 BC00032 VJ=100.00  +MOVJ EC00032 VJ=100.00
MOVJ C00033 BC00033 VJ=100.00  +MOVJ EC00033 VJ=100.00
MOVJ C00034 BC00034 VJ=100.00  +MOVJ EC00034 VJ=100.00
MOVJ C00035 BC00035 VJ=100.00  +MOVJ EC00035 VJ=100.00
COMM 'Path S4675
COMM SFTOF3D
COMM MOVJ C00036 BC00036 VJ=100.00  +MOVJ EC00036 VJ=100.00
COMM PAUSE
COMM MOVL C00037 BC00037 V=800.0  +MOVJ EC00037 VJ=100.00
COMM SMOVL C00038 BC00038 V=166.7  +MOVJ EC00038
COMM SREFP 3 C00039 BC00039  +REFP EC00039
COMM CALL JOB:SEARCH-R1-S13D
COMM SET P041 P006
COMM SFTON3D P041
COMM SMOVL C00040 BC00040 V=166.7  +MOVJ EC00040
COMM SMOVL C00041 BC00041 V=166.7  +MOVJ EC00041
COMM SREFP 3 C00042 BC00042  +REFP EC00042
COMM CALL JOB:SEARCH-R1-S13D
COMM SET P041 P006
COMM SFTON3D P041
COMM SMOVL C00043 BC00043 V=166.7  +MOVJ EC00043
COMM SMOVL C00044 BC00044 V=166.7  +MOVJ EC00044
COMM MOVL C00045 BC00045 V=1000.0  +MOVJ EC00045 VJ=100.00
COMM 'EndPath S4675
COMM 'Path S4676
COMM SFTOF3D
COMM MOVJ C00046 BC00046 VJ=100.00  +MOVJ EC00046 VJ=100.00
COMM MOVL C00047 BC00047 V=800.0  +MOVJ EC00047 VJ=100.00
COMM SMOVL C00048 BC00048 V=166.7  +MOVJ EC00048
COMM SREFP 3 C00049 BC00049  +REFP EC00049
COMM CALL JOB:SEARCH-R1-S13D
COMM SET P042 P006
COMM SFTON3D P042
COMM SMOVL C00050 BC00050 V=166.7  +MOVJ EC00050
COMM SMOVL C00051 BC00051 V=166.7  +MOVJ EC00051
COMM SREFP 3 C00052 BC00052  +REFP EC00052
COMM CALL JOB:SEARCH-R1-S13D
COMM SET P042 P006
COMM SFTON3D P042
COMM SMOVL C00053 BC00053 V=166.7  +MOVJ EC00053
COMM SMOVL C00054 BC00054 V=166.7  +MOVJ EC00054
COMM MOVL C00055 BC00055 V=1000.0  +MOVJ EC00055 VJ=100.00
COMM 'EndPath S4676
COMM MOVJ C00056 BC00056 VJ=100.00  +MOVJ EC00056 VJ=100.00
COMM PAUSE
MOVJ C00057 BC00057 VJ=100.00  +MOVJ EC00057 VJ=100.00
'Path S4677
SFTOF3D
MOVJ C00058 BC00058 VJ=100.00  +MOVJ EC00058 VJ=100.00
MOVL C00059 BC00059 V=800.0  +MOVJ EC00059 VJ=100.00
SMOVL C00060 BC00060 V=166.7  +MOVJ EC00060
SREFP 3 C00061 BC00061  +REFP EC00061
CALL JOB:SEARCH-R1-S13D
SET P023 P006
SFTON3D P023
SMOVL C00062 BC00062 V=166.7  +MOVJ EC00062
SREFP 3 C00063 BC00063  +REFP EC00063
CALL JOB:SEARCH-R1-S13D
SET P023 P006
SFTON3D P023
SMOVL C00064 BC00064 V=166.7  +MOVJ EC00064
SMOVL C00065 BC00065 V=166.7  +MOVJ EC00065
SREFP 3 C00066 BC00066  +REFP EC00066
CALL JOB:SEARCH-R1-S13D
SET P023 P006
SFTON3D P023
SMOVL C00067 BC00067 V=166.7  +MOVJ EC00067
MOVL C00068 BC00068 V=1000.0  +MOVJ EC00068 VJ=100.00
'EndPath S4677
'Path S4678
SFTOF3D
MOVJ C00069 BC00069 VJ=100.00  +MOVJ EC00069 VJ=100.00
MOVL C00070 BC00070 V=800.0  +MOVJ EC00070 VJ=100.00
SMOVL C00071 BC00071 V=166.7  +MOVJ EC00071
SREFP 3 C00072 BC00072  +REFP EC00072
CALL JOB:SEARCH-R1-S13D
SET P024 P006
SFTON3D P024
SMOVL C00073 BC00073 V=166.7  +MOVJ EC00073
SREFP 3 C00074 BC00074  +REFP EC00074
CALL JOB:SEARCH-R1-S13D
SET P024 P006
SFTON3D P024
SMOVL C00075 BC00075 V=166.7  +MOVJ EC00075
MOVL C00076 BC00076 V=1000.0  +MOVJ EC00076 VJ=100.00
'EndPath S4678
MOVJ C00077 BC00077 VJ=100.00  +MOVJ EC00077 VJ=100.00
MOVJ C00078 BC00078 VJ=100.00  +MOVJ EC00078 VJ=100.00
'Path S4679
SFTOF3D
MOVJ C00079 BC00079 VJ=100.00  +MOVJ EC00079 VJ=100.00
MOVL C00080 BC00080 V=800.0  +MOVJ EC00080 VJ=100.00
SMOVL C00081 BC00081 V=166.7  +MOVJ EC00081
SREFP 3 C00082 BC00082  +REFP EC00082
CALL JOB:SEARCH-R1-S13D
SET P025 P006
SFTON3D P025
SMOVL C00083 BC00083 V=166.7  +MOVJ EC00083
SREFP 3 C00084 BC00084  +REFP EC00084
CALL JOB:SEARCH-R1-S13D
SET P025 P006
SFTON3D P025
SMOVL C00085 BC00085 V=166.7  +MOVJ EC00085
MOVL C00086 BC00086 V=1000.0  +MOVJ EC00086 VJ=100.00
'EndPath S4679
'Path S4680
SFTOF3D
MOVJ C00087 BC00087 VJ=100.00  +MOVJ EC00087 VJ=100.00
MOVL C00088 BC00088 V=800.0  +MOVJ EC00088 VJ=100.00
SMOVL C00089 BC00089 V=166.7  +MOVJ EC00089
SREFP 3 C00090 BC00090  +REFP EC00090
CALL JOB:SEARCH-R1-S13D
SET P026 P006
SFTON3D P026
SMOVL C00091 BC00091 V=166.7  +MOVJ EC00091
SMOVL C00092 BC00092 V=166.7  +MOVJ EC00092
SREFP 3 C00093 BC00093  +REFP EC00093
CALL JOB:SEARCH-R1-S13D
SET P026 P006
SFTON3D P026
SMOVL C00094 BC00094 V=166.7  +MOVJ EC00094
MOVL C00095 BC00095 V=1000.0  +MOVJ EC00095 VJ=100.00
'EndPath S4680
MOVJ C00096 BC00096 VJ=100.00  +MOVJ EC00096 VJ=100.00
'Up
MOVJ C00097 BC00097 VJ=100.00  +MOVJ EC00097 VJ=100.00
MOVJ C00098 BC00098 VJ=100.00  +MOVJ EC00098 VJ=100.00
'Path S4681
SFTOF3D
MOVJ C00099 BC00099 VJ=100.00  +MOVJ EC00099 VJ=100.00
MOVL C00100 BC00100 V=800.0  +MOVJ EC00100 VJ=100.00
SMOVL C00101 BC00101 V=166.7  +MOVJ EC00101
SREFP 3 C00102 BC00102  +REFP EC00102
CALL JOB:SEARCH-R1-S13D
SET P031 P006
SFTON3D P031
SMOVL C00103 BC00103 V=166.7  +MOVJ EC00103
SREFP 3 C00104 BC00104  +REFP EC00104
CALL JOB:SEARCH-R1-S13D
SET P031 P006
SFTON3D P031
SMOVL C00105 BC00105 V=166.7  +MOVJ EC00105
SMOVL C00106 BC00106 V=166.7  +MOVJ EC00106
SREFP 3 C00107 BC00107  +REFP EC00107
CALL JOB:SEARCH-R1-S13D
SET P031 P006
SFTON3D P031
SMOVL C00108 BC00108 V=166.7  +MOVJ EC00108
MOVL C00109 BC00109 V=800.0  +MOVJ EC00109 VJ=100.00
MOVL C00110 BC00110 V=1000.0  +MOVJ EC00110 VJ=100.00
'EndPath S4681
MOVJ C00111 BC00111 VJ=100.00  +MOVJ EC00111 VJ=100.00
'Path S4682
SFTOF3D
MOVJ C00112 BC00112 VJ=100.00  +MOVJ EC00112 VJ=100.00
MOVL C00113 BC00113 V=800.0  +MOVJ EC00113 VJ=100.00
SMOVL C00114 BC00114 V=166.7  +MOVJ EC00114
SREFP 3 C00115 BC00115  +REFP EC00115
CALL JOB:SEARCH-R1-S13D
SET P032 P006
SFTON3D P032
SMOVL C00116 BC00116 V=166.7  +MOVJ EC00116
SREFP 3 C00117 BC00117  +REFP EC00117
CALL JOB:SEARCH-R1-S13D
SET P032 P006
SFTON3D P032
SMOVL C00118 BC00118 V=166.7  +MOVJ EC00118
SMOVL C00119 BC00119 V=166.7  +MOVJ EC00119
SREFP 3 C00120 BC00120  +REFP EC00120
CALL JOB:SEARCH-R1-S13D
SET P032 P006
SFTON3D P032
SMOVL C00121 BC00121 V=166.7  +MOVJ EC00121
MOVL C00122 BC00122 V=1000.0  +MOVJ EC00122 VJ=100.00
'EndPath S4682
MOVJ C00123 BC00123 VJ=100.00  +MOVJ EC00123 VJ=100.00
'Path S4683
SFTOF3D
MOVJ C00124 BC00124 VJ=100.00  +MOVJ EC00124 VJ=100.00
MOVL C00125 BC00125 V=800.0  +MOVJ EC00125 VJ=100.00
SMOVL C00126 BC00126 V=166.7  +MOVJ EC00126
SREFP 3 C00127 BC00127  +REFP EC00127
CALL JOB:SEARCH-R1-S13D
SET P033 P006
SFTON3D P033
SMOVL C00128 BC00128 V=166.7  +MOVJ EC00128
SREFP 3 C00129 BC00129  +REFP EC00129
CALL JOB:SEARCH-R1-S13D
SET P033 P006
SFTON3D P033
SMOVL C00130 BC00130 V=166.7  +MOVJ EC00130
SMOVL C00131 BC00131 V=166.7  +MOVJ EC00131
SREFP 3 C00132 BC00132  +REFP EC00132
CALL JOB:SEARCH-R1-S13D
SET P033 P006
SFTON3D P033
SMOVL C00133 BC00133 V=166.7  +MOVJ EC00133
MOVL C00134 BC00134 V=1000.0  +MOVJ EC00134 VJ=100.00
MOVL C00135 BC00135 V=1000.0  +MOVJ EC00135 VJ=100.00
'EndPath S4683
MOVJ C00136 BC00136 VJ=100.00  +MOVJ EC00136 VJ=100.00
'Path S4684
SFTOF3D
MOVJ C00137 BC00137 VJ=100.00  +MOVJ EC00137 VJ=100.00
MOVL C00138 BC00138 V=800.0  +MOVJ EC00138 VJ=100.00
SMOVL C00139 BC00139 V=166.7  +MOVJ EC00139
SREFP 3 C00140 BC00140  +REFP EC00140
CALL JOB:SEARCH-R1-S13D
SET P034 P006
SFTON3D P034
SMOVL C00141 BC00141 V=166.7  +MOVJ EC00141
SREFP 3 C00142 BC00142  +REFP EC00142
CALL JOB:SEARCH-R1-S13D
SET P034 P006
SFTON3D P034
SMOVL C00143 BC00143 V=166.7  +MOVJ EC00143
SMOVL C00144 BC00144 V=166.7  +MOVJ EC00144
SREFP 3 C00145 BC00145  +REFP EC00145
CALL JOB:SEARCH-R1-S13D
SET P034 P006
SFTON3D P034
SMOVL C00146 BC00146 V=166.7  +MOVJ EC00146
MOVL C00147 BC00147 V=800.0  +MOVJ EC00147 VJ=100.00
MOVL C00148 BC00148 V=1000.0  +MOVJ EC00148 VJ=100.00
MOVL C00149 BC00149 V=1000.0  +MOVJ EC00149 VJ=100.00
'EndPath S4684
MOVJ C00150 BC00150 VJ=100.00  +MOVJ EC00150 VJ=100.00
'Path S4685
SFTOF3D
MOVJ C00151 BC00151 VJ=100.00  +MOVJ EC00151 VJ=100.00
MOVL C00152 BC00152 V=800.0  +MOVJ EC00152 VJ=100.00
SMOVL C00153 BC00153 V=166.7  +MOVJ EC00153
SREFP 3 C00154 BC00154  +REFP EC00154
CALL JOB:SEARCH-R1-S13D
SET P035 P006
SFTON3D P035
SMOVL C00155 BC00155 V=166.7  +MOVJ EC00155
SMOVL C00156 BC00156 V=166.7  +MOVJ EC00156
SREFP 3 C00157 BC00157  +REFP EC00157
CALL JOB:SEARCH-R1-S13D
SET P035 P006
SFTON3D P035
SMOVL C00158 BC00158 V=166.7  +MOVJ EC00158
SMOVL C00159 BC00159 V=166.7  +MOVJ EC00159
SREFP 3 C00160 BC00160  +REFP EC00160
CALL JOB:SEARCH-R1-S13D
SET P035 P006
SFTON3D P035
SMOVL C00161 BC00161 V=166.7  +MOVJ EC00161
MOVL C00162 BC00162 V=1000.0  +MOVJ EC00162 VJ=100.00
'EndPath S4685
MOVJ C00163 BC00163 VJ=100.00  +MOVJ EC00163 VJ=100.00
'Path S4686
SFTOF3D
MOVJ C00164 BC00164 VJ=100.00  +MOVJ EC00164 VJ=100.00
MOVL C00165 BC00165 V=800.0  +MOVJ EC00165 VJ=100.00
SMOVL C00166 BC00166 V=166.7  +MOVJ EC00166
SREFP 3 C00167 BC00167  +REFP EC00167
CALL JOB:SEARCH-R1-S13D
SET P036 P006
SFTON3D P036
SMOVL C00168 BC00168 V=166.7  +MOVJ EC00168
SMOVL C00169 BC00169 V=166.7  +MOVJ EC00169
SREFP 3 C00170 BC00170  +REFP EC00170
CALL JOB:SEARCH-R1-S13D
SET P036 P006
SFTON3D P036
SMOVL C00171 BC00171 V=166.7  +MOVJ EC00171
SMOVL C00172 BC00172 V=166.7  +MOVJ EC00172
SREFP 3 C00173 BC00173  +REFP EC00173
CALL JOB:SEARCH-R1-S13D
SET P036 P006
SFTON3D P036
SMOVL C00174 BC00174 V=166.7  +MOVJ EC00174
MOVL C00175 BC00175 V=1000.0  +MOVJ EC00175 VJ=100.00
'EndPath S4686
MOVJ C00176 BC00176 VJ=100.00  +MOVJ EC00176 VJ=100.00
'Path S4687
SFTOF3D
MOVJ C00177 BC00177 VJ=100.00  +MOVJ EC00177 VJ=100.00
MOVL C00178 BC00178 V=800.0  +MOVJ EC00178 VJ=100.00
SMOVL C00179 BC00179 V=166.7  +MOVJ EC00179
SREFP 3 C00180 BC00180  +REFP EC00180
CALL JOB:SEARCH-R1-S13D
SET P037 P006
SFTON3D P037
SMOVL C00181 BC00181 V=166.7  +MOVJ EC00181
SMOVL C00182 BC00182 V=166.7  +MOVJ EC00182
SREFP 3 C00183 BC00183  +REFP EC00183
CALL JOB:SEARCH-R1-S13D
SET P037 P006
SFTON3D P037
SMOVL C00184 BC00184 V=166.7  +MOVJ EC00184
SMOVL C00185 BC00185 V=166.7  +MOVJ EC00185
SREFP 3 C00186 BC00186  +REFP EC00186
CALL JOB:SEARCH-R1-S13D
SET P037 P006
SFTON3D P037
SMOVL C00187 BC00187 V=166.7  +MOVJ EC00187
MOVL C00188 BC00188 V=1000.0  +MOVJ EC00188 VJ=100.00
'EndPath S4687
MOVJ C00189 BC00189 VJ=100.00  +MOVJ EC00189 VJ=100.00
'Path S4688
SFTOF3D
MOVJ C00190 BC00190 VJ=100.00  +MOVJ EC00190 VJ=100.00
MOVL C00191 BC00191 V=800.0  +MOVJ EC00191 VJ=100.00
SMOVL C00192 BC00192 V=166.7  +MOVJ EC00192
SREFP 3 C00193 BC00193  +REFP EC00193
CALL JOB:SEARCH-R1-S13D
SET P038 P006
SFTON3D P038
SMOVL C00194 BC00194 V=166.7  +MOVJ EC00194
SMOVL C00195 BC00195 V=166.7  +MOVJ EC00195
SREFP 3 C00196 BC00196  +REFP EC00196
CALL JOB:SEARCH-R1-S13D
SET P038 P006
SFTON3D P038
SMOVL C00197 BC00197 V=166.7  +MOVJ EC00197
SMOVL C00198 BC00198 V=166.7  +MOVJ EC00198
SREFP 3 C00199 BC00199  +REFP EC00199
CALL JOB:SEARCH-R1-S13D
SET P038 P006
SFTON3D P038
SMOVL C00200 BC00200 V=166.7  +MOVJ EC00200
MOVL C00201 BC00201 V=800.0  +MOVJ EC00201 VJ=100.00
MOVL C00202 BC00202 V=1000.0  +MOVJ EC00202 VJ=100.00
'EndPath S4688
MOVJ C00203 BC00203 VJ=100.00  +MOVJ EC00203 VJ=100.00
'Path S4689
SFTOF3D
MOVJ C00204 BC00204 VJ=100.00  +MOVJ EC00204 VJ=100.00
MOVL C00205 BC00205 V=800.0  +MOVJ EC00205 VJ=100.00
SMOVL C00206 BC00206 V=166.7  +MOVJ EC00206
SREFP 3 C00207 BC00207  +REFP EC00207
CALL JOB:SEARCH-R1-S13D
SET P039 P006
SFTON3D P039
SMOVL C00208 BC00208 V=166.7  +MOVJ EC00208
SMOVL C00209 BC00209 V=166.7  +MOVJ EC00209
SREFP 3 C00210 BC00210  +REFP EC00210
CALL JOB:SEARCH-R1-S13D
SET P039 P006
SFTON3D P039
SMOVL C00211 BC00211 V=166.7  +MOVJ EC00211
SMOVL C00212 BC00212 V=166.7  +MOVJ EC00212
SREFP 3 C00213 BC00213  +REFP EC00213
CALL JOB:SEARCH-R1-S13D
SET P039 P006
SFTON3D P039
SMOVL C00214 BC00214 V=166.7  +MOVJ EC00214
MOVL C00215 BC00215 V=1000.0  +MOVJ EC00215 VJ=100.00
'EndPath S4689
'Path S4690
SFTOF3D
MOVJ C00216 BC00216 VJ=100.00  +MOVJ EC00216 VJ=100.00
MOVL C00217 BC00217 V=800.0  +MOVJ EC00217 VJ=100.00
SMOVL C00218 BC00218 V=166.7  +MOVJ EC00218
SREFP 3 C00219 BC00219  +REFP EC00219
CALL JOB:SEARCH-R1-S13D
SET P040 P006
SFTON3D P040
SMOVL C00220 BC00220 V=166.7  +MOVJ EC00220
SREFP 3 C00221 BC00221  +REFP EC00221
CALL JOB:SEARCH-R1-S13D
SET P040 P006
SFTON3D P040
SMOVL C00222 BC00222 V=166.7  +MOVJ EC00222
MOVL C00223 BC00223 V=1000.0  +MOVJ EC00223 VJ=100.00
'EndPath S4690
'Path W4691
SFTOF3D
SFTON3D P039
MOVJ C00224 BC00224 VJ=100.00  +MOVJ EC00224 VJ=100.00
SMOVL C00225 BC00225 V=800.0  +MOVJ EC00225
SMOVL C00226 BC00226 V=166.7 PL=0  +MOVJ EC00226
MACRO1 MJ#(0) ARGF21
ARCON
SMOVL C00227 BC00227 V=7.5  +MOVJ EC00227
SFTON3D P040
SMOVL C00228 BC00228 V=7.5  +MOVJ EC00228
SMOVL C00229 BC00229 V=7.5  +MOVJ EC00229
ARCOF
SMOVL C00230 BC00230 V=800.0  +MOVJ EC00230
SMOVL C00231 BC00231 V=1000.0  +MOVJ EC00231
SFTOF3D
'EndPath W4691
'Path W4692
SFTOF3D
SFTON3D P037
MOVJ C00232 BC00232 VJ=100.00  +MOVJ EC00232 VJ=100.00
MOVJ C00233 BC00233 VJ=100.00  +MOVJ EC00233 VJ=100.00
MOVJ C00234 BC00234 VJ=100.00  +MOVJ EC00234 VJ=100.00
SMOVL C00235 BC00235 V=800.0  +MOVJ EC00235
SMOVL C00236 BC00236 V=166.7 PL=0  +MOVJ EC00236
MACRO1 MJ#(0) ARGF14
ARCON
SMOVL C00237 BC00237 V=10.0  +MOVJ EC00237
SMOVL C00238 BC00238 V=10.0  +MOVJ EC00238
SMOVL C00239 BC00239 V=10.0  +MOVJ EC00239
SFTON3D P038
SMOVL C00240 BC00240 V=10.0  +MOVJ EC00240
SMOVL C00241 BC00241 V=10.0  +MOVJ EC00241
ARCOF
SMOVL C00242 BC00242 V=800.0  +MOVJ EC00242
SMOVL C00243 BC00243 V=1000.0  +MOVJ EC00243
SFTOF3D
'EndPath W4692
MOVJ C00244 BC00244 VJ=100.00  +MOVJ EC00244 VJ=100.00
'Path W4693
SFTOF3D
SFTON3D P035
MOVJ C00245 BC00245 VJ=100.00  +MOVJ EC00245 VJ=100.00
MOVJ C00246 BC00246 VJ=100.00  +MOVJ EC00246 VJ=100.00
SMOVL C00247 BC00247 V=800.0  +MOVJ EC00247
SMOVL C00248 BC00248 V=166.7 PL=0  +MOVJ EC00248
ARCON
SMOVL C00249 BC00249 V=10.0  +MOVJ EC00249
SMOVL C00250 BC00250 V=10.0  +MOVJ EC00250
SMOVL C00251 BC00251 V=10.0  +MOVJ EC00251
SFTON3D P036
SMOVL C00252 BC00252 V=10.0  +MOVJ EC00252
SMOVL C00253 BC00253 V=10.0  +MOVJ EC00253
ARCOF
SMOVL C00254 BC00254 V=800.0  +MOVJ EC00254
SMOVL C00255 BC00255 V=1000.0  +MOVJ EC00255
SMOVL C00256 BC00256 V=1000.0  +MOVJ EC00256
SFTOF3D
'EndPath W4693
MOVJ C00257 BC00257 VJ=100.00  +MOVJ EC00257 VJ=100.00
'Path W4694
SFTOF3D
SFTON3D P033
MOVJ C00258 BC00258 VJ=100.00  +MOVJ EC00258 VJ=100.00
SMOVL C00259 BC00259 V=800.0  +MOVJ EC00259
SMOVL C00260 BC00260 V=166.7 PL=0  +MOVJ EC00260
MACRO1 MJ#(0) ARGF9
ARCON
SMOVL C00261 BC00261 V=10.0  +MOVJ EC00261
SFTON3D P034
SMOVL C00262 BC00262 V=10.0  +MOVJ EC00262
SMOVL C00263 BC00263 V=10.0  +MOVJ EC00263
ARCOF
SMOVL C00264 BC00264 V=800.0  +MOVJ EC00264
SMOVL C00265 BC00265 V=1000.0  +MOVJ EC00265
SMOVL C00266 BC00266 V=1000.0  +MOVJ EC00266
SFTOF3D
'EndPath W4694
MOVJ C00267 BC00267 VJ=100.00  +MOVJ EC00267 VJ=100.00
'Path W4695
SFTOF3D
SFTON3D P032
MOVJ C00268 BC00268 VJ=100.00  +MOVJ EC00268 VJ=100.00
MOVJ C00269 BC00269 VJ=100.00  +MOVJ EC00269 VJ=100.00
SMOVL C00270 BC00270 V=800.0  +MOVJ EC00270
SMOVL C00271 BC00271 V=166.7 PL=0  +MOVJ EC00271
ARCON
SMOVL C00272 BC00272 V=10.5  +MOVJ EC00272
SFTON3D P031
SMOVL C00273 BC00273 V=10.5  +MOVJ EC00273
SMOVL C00274 BC00274 V=10.5  +MOVJ EC00274
ARCOF
SMOVL C00275 BC00275 V=800.0  +MOVJ EC00275
SMOVL C00276 BC00276 V=1000.0  +MOVJ EC00276
SFTOF3D
'EndPath W4695
MOVJ C00277 BC00277 VJ=100.00  +MOVJ EC00277 VJ=100.00
MOVJ C00278 BC00278 VJ=100.00  +MOVJ EC00278 VJ=100.00
'Down
MOVJ C00279 BC00279 VJ=100.00  +MOVJ EC00279 VJ=100.00
'Path W4696
SFTOF3D
SFTON3D P026
MOVJ C00280 BC00280 VJ=100.00  +MOVJ EC00280 VJ=100.00
SMOVL C00281 BC00281 V=800.0  +MOVJ EC00281
SMOVL C00282 BC00282 V=150.0 PL=0  +MOVJ EC00282
MACRO1 MJ#(0) ARGF22
ARCON
SWVON WEV#(108)
SMOVC C00283 BC00283 V=10.0  +MOVJ EC00283
SMOVC C00284 BC00284 V=10.0  +MOVJ EC00284
SMOVC C00285 BC00285 V=10.0  +MOVJ EC00285
SFTON3D P025
SMOVC C00286 BC00286 V=10.0  +MOVJ EC00286
SMOVC C00287 BC00287 V=10.0  +MOVJ EC00287
SMOVC C00288 BC00288 V=10.0  +MOVJ EC00288
SMOVL C00289 BC00289 V=10.0  +MOVJ EC00289
ARCOF
SWVOF
SMOVL C00290 BC00290 V=800.0  +MOVJ EC00290
SMOVL C00291 BC00291 V=1000.0  +MOVJ EC00291
SFTOF3D
'EndPath W4696
MOVJ C00292 BC00292 VJ=100.00  +MOVJ EC00292 VJ=100.00
MOVJ C00293 BC00293 VJ=100.00  +MOVJ EC00293 VJ=100.00
MOVJ C00294 BC00294 VJ=100.00  +MOVJ EC00294 VJ=100.00
MOVJ C00295 BC00295 VJ=100.00  +MOVJ EC00295 VJ=100.00
'Path W4697
SFTOF3D
SFTON3D P022
MOVJ C00296 BC00296 VJ=100.00  +MOVJ EC00296 VJ=100.00
MOVJ C00297 BC00297 VJ=100.00  +MOVJ EC00297 VJ=100.00
SFTON3D P022
SMOVL C00298 BC00298 V=800.0  +MOVJ EC00298
SMOVL C00299 BC00299 V=166.7 PL=0  +MOVJ EC00299
MACRO1 MJ#(0) ARGF9
ARCON
SMOVL C00300 BC00300 V=10.0  +MOVJ EC00300
SMOVL C00301 BC00301 V=10.0  +MOVJ EC00301
SMOVL C00302 BC00302 V=10.0  +MOVJ EC00302
SMOVL C00303 BC00303 V=10.0  +MOVJ EC00303
SMOVL C00304 BC00304 V=10.0  +MOVJ EC00304
SMOVL C00305 BC00305 V=10.0  +MOVJ EC00305
SMOVL C00306 BC00306 V=10.0  +MOVJ EC00306
SMOVL C00307 BC00307 V=10.0  +MOVJ EC00307
SMOVL C00308 BC00308 V=10.0  +MOVJ EC00308
ARCOF
SMOVL C00309 BC00309 V=800.0  +MOVJ EC00309
SMOVL C00310 BC00310 V=1000.0  +MOVJ EC00310
SFTOF3D
'EndPath W4697
'Path W4698
SFTOF3D
SFTON3D P021
SFTOF3D
'EndPath W4698
MOVJ C00311 BC00311 VJ=100.00  +MOVJ EC00311 VJ=100.00
'Path W4699
SFTOF3D
SFTON3D P020
MOVJ C00312 BC00312 VJ=100.00  +MOVJ EC00312 VJ=100.00
SMOVL C00313 BC00313 V=800.0  +MOVJ EC00313
SMOVL C00314 BC00314 V=150.0 PL=0  +MOVJ EC00314
ARCON
SMOVL C00315 BC00315 V=8.3  +MOVJ EC00315
ARCOF
SMOVL C00316 BC00316 V=800.0  +MOVJ EC00316
SFTOF3D
'EndPath W4699
MOVJ C00317 BC00317 VJ=100.00  +MOVJ EC00317 VJ=100.00
MOVJ C00318 BC00318 VJ=100.00  +MOVJ EC00318 VJ=100.00
MOVJ C00319 BC00319 VJ=100.00  +MOVJ EC00319 VJ=100.00
MOVJ C00320 BC00320 VJ=100.00  +MOVJ EC00320 VJ=100.00
'Path W4700
SFTOF3D
SFTON3D P023
MOVJ C00321 BC00321 VJ=100.00  +MOVJ EC00321 VJ=100.00
SMOVL C00322 BC00322 V=800.0  +MOVJ EC00322
'POSPAWANE
SMOVC C00323 BC00323 V=150.0 PL=0  +MOVJ EC00323
MACRO1 MJ#(0) ARGF22
ARCON
SWVON WEV#(108)
SMOVC C00324 BC00324 V=10.0  +MOVJ EC00324
ARCON
SMOVC C00325 BC00325 V=10.0  +MOVJ EC00325
SFTON3D P024
ARCON
SMOVC C00326 BC00326 V=10.0  +MOVJ EC00326
SMOVL C00327 BC00327 V=10.0  +MOVJ EC00327
ARCOF
SWVOF
SMOVL C00328 BC00328 V=800.0  +MOVJ EC00328
SMOVL C00329 BC00329 V=1000.0  +MOVJ EC00329
SFTOF3D
'EndPath W4700
MOVJ C00330 BC00330 VJ=100.00  +MOVJ EC00330 VJ=100.00
'jakie searche do takicj spoin?
'kamera
MOVJ C00331 BC00331 VJ=100.00  +MOVJ EC00331 VJ=100.00
MOVJ C00332 BC00332 VJ=100.00  +MOVJ EC00332 VJ=100.00
'Path W4701
SFTOF3D
SFTON3D P041
MOVJ C00333 BC00333 VJ=100.00  +MOVJ EC00333 VJ=100.00
COMM PAUSE
COMM SMOVL C00334 BC00334 V=800.0  +MOVJ EC00334
COMM SMOVL C00335 BC00335 V=150.0 PL=0  +MOVJ EC00335
COMM MACRO1 MJ#(0) ARGF9
COMM ARCON
COMM SMOVL C00336 BC00336 V=11.7  +MOVJ EC00336
COMM ARCOF
COMM SMOVL C00337 BC00337 V=800.0  +MOVJ EC00337
COMM SMOVL C00338 BC00338 V=1000.0  +MOVJ EC00338
COMM SFTOF3D
COMM 'EndPath W4708
COMM 'Path W4709
COMM SFTOF3D
COMM SFTON3D P042
COMM MOVJ C00339 BC00339 VJ=100.00  +MOVJ EC00339 VJ=100.00
COMM SMOVL C00340 BC00340 V=800.0  +MOVJ EC00340
COMM SMOVL C00341 BC00341 V=150.0 PL=0  +MOVJ EC00341
COMM ARCON
COMM SMOVL C00342 BC00342 V=11.7  +MOVJ EC00342
COMM ARCOF
COMM SMOVL C00343 BC00343 V=800.0  +MOVJ EC00343
COMM SMOVL C00344 BC00344 V=1000.0  +MOVJ EC00344
COMM SMOVL C00345 BC00345 V=1000.0  +MOVJ EC00345
SFTOF3D
'EndPath W4709
'Path W4710
SFTOF3D
SMOVL C00346 BC00346 V=333.3  +MOVJ EC00346
MOVJ C00347 BC00347 VJ=100.00  +MOVJ EC00347 VJ=100.00
MOVJ C00348 BC00348 VJ=100.00  +MOVJ EC00348 VJ=100.00
MOVL C00349 BC00349 V=800.0  +MOVJ EC00349 VJ=100.00
SMOVL C00350 BC00350 V=166.7 PL=0  +MOVJ EC00350
MACRO1 MJ#(0) ARGF20
ARCON
SMOVL C00351 BC00351 V=6.7  +MOVJ EC00351
SMOVL C00352 BC00352 V=6.7  +MOVJ EC00352
SMOVL C00353 BC00353 V=6.7  +MOVJ EC00353
ARCOF
MOVL C00354 BC00354 V=800.0  +MOVJ EC00354 VJ=100.00
MOVL C00355 BC00355 V=1000.0  +MOVJ EC00355 VJ=100.00
'EndPath W4710
MOVJ C00356 BC00356 VJ=100.00  +MOVJ EC00356 VJ=100.00
MOVJ C00357 BC00357 VJ=100.00  +MOVJ EC00357 VJ=100.00
MOVJ C00358 BC00358 VJ=100.00  +MOVJ EC00358 VJ=100.00
'68,69
'
END
